Omron CX-Programmer project NewProject (CX-Programmer 9.75)

# PLC NewPLC1: CP1H XA

## Program SCL_Convert_Program (cyclic task 0)

### Section Section_1

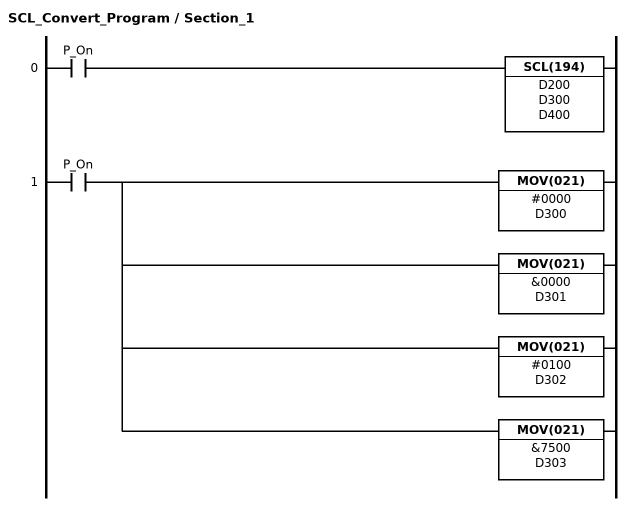
; rung 0
LD P_On
SCL(194) D200 D300 D400
; rung 1
LD P_On
MOV(021) #0000 D300
MOV(021) &0000 D301
MOV(021) #0100 D302
MOV(021) &7500 D303

### Section END
; rung 0
END(001)